// TIA Portal V18 export
TYPE "LGasp_typeSyncAttuatore"
// stored: IsFailsafeCompliant false
   STRUCT
      qsync { ExternalAccessible := 'False'; ExternalVisible := 'False'; ExternalWritable := 'False'} : LReal;   // Quota di set posizione nel caso di un asse
      cmdsync { ExternalAccessible := 'False'; ExternalVisible := 'False'; ExternalWritable := 'False'} : Bool;   // Comando set posizione(sync) nel caso di un asse
   END_STRUCT;
END_TYPE
